FUNCTION_BLOCK T_CollectionBase EXTENDS T_NamedBase
VAR
    _items : ARRAY[0..(COLLECTION_MAX_SIZE-1)] OF I_InterfaceBase;
    _cnt : UDINT;
END_VAR
VAR CONSTANT
    COLLECTION_MAX_SIZE : UDINT := Parameters_PackML_Base.COLLECTION_MAX_SIZE;
END_VAR

METHOD PRIVATE addInSpareSlot : BOOL
VAR_INPUT
	Item : I_InterfaceBase;
END_VAR
IF Count >= COLLECTION_MAX_SIZE THEN
	LogError('cannot addInSpareSlot : no space.');
	RETURN;
END_IF
	
_items[Count] := Item;
Count := Count + 1;
addInSpareSlot := TRUE;
END_METHOD

METHOD INTERNAL AddItem : BOOL
VAR_INPUT
  newItem : I_InterfaceBase;
END_VAR
IF newItem = 0 THEN
	LogError( 'Cannot AddComponent invalid ref' );
	RETURN;
END_IF

IF HasItem( Item := newItem ) THEN
	LogWarning( 'Component already in collection.' );
	RETURN;
END_IF

AddItem := addInSpareSlot( Item := newItem );
END_METHOD

METHOD ClearGroup // clears the group down
MEMSET(ADR(_items), 0 , SIZEOF(_items));
_cnt := 0;
LogDebug('ClearGroup() called.');
END_METHOD

PROPERTY Count : UDINT
GET
Count := _cnt;
END_GET
SET // PRIVATE
_cnt := Count;
END_SET
END_PROPERTY

METHOD PRIVATE HasItem : BOOL
VAR_INPUT
	Item : I_InterfaceBase;
END_VAR
VAR 
	i : UDINT;
END_VAR
IF Count >= COLLECTION_MAX_SIZE THEN
	LogWarning('Count Exceed Collection Max Size');
	RETURN;
END_IF

FOR i := 0 TO Count DO
	
	IF _items[i] = 0 THEN
		EXIT; // exit for loop
	END_IF
	
	IF _items[i] = Item THEN
		HasItem := TRUE;
		RETURN;
		
	END_IF
	
END_FOR
END_METHOD

METHOD INTERNAL TryGetItem: BOOL
VAR_INPUT
	index : UDINT;
END_VAR
VAR_OUTPUT
	item : I_InterfaceBase;
END_VAR
IF index > (COLLECTION_MAX_SIZE-1) THEN
	LogError( 'cannot GetDrive, index out of bounds' );
	RETURN;
END_IF

IF index > Count THEN
	LogError( 'cannot GetDrive, index > (Count - 1) ' );
	RETURN;
END_IF

item := _items[index];
TryGetItem := item <> 0;
END_METHOD

END_FUNCTION_BLOCK

(* stored: Version 1.1.0.1, ProductVersion 3.1.4024.12
   POU T_CollectionBase: Id {91f145eb-820d-4f7a-9926-40255bcc85a0}, SpecialFunc None
   Folder Private: Id {b567f85d-3012-43a8-97ff-301076c39f5d}
   Method addInSpareSlot: Id {8c3d3185-0175-4738-9c73-0037742ace98}
   Method AddItem: Id {694024fe-c5ed-4d58-959e-acc65fd5108c}
   Method ClearGroup: Id {33765d55-9a26-4942-8a3f-e0d7968dad36}
   Property Count: Id {8e6ae03a-8f5c-414d-ab3f-cfcd3d9da8a8}
   Get Get: Id {6eadc8ba-599e-4f96-a78c-8d7470a97016}
   Set Set: Id {766f63da-f17d-49ca-a39f-c9fa2a12c25c}
   Method HasItem: Id {3ce85fba-0a5e-4fa1-9c6a-844b57d80979}
   Method TryGetItem: Id {4079f152-eedc-41b9-985e-004de6f818fa} *)
